FUNCTION_BLOCK fbLightControlV2
		
VAR_INPUT
	bButtonhoofdFunctie				: BOOL;
	bButton2				: BOOL;
	bForceOff			: BOOL;
	bForceOn			: BOOL;

END_VAR
VAR_OUTPUT
	bLight1				: BOOL;
	bLight2				: BOOL;	
	
END_VAR
VAR
	InputTriggerHoofd		: R_trig; 
	InputTrigger2		: R_trig; 
	test:BOOL;
	iCaseVar			:UINT; 
	

	
END_VAR


// This is the first version, ignoring all debounce timers and other issues 
// Base function is a to allow switching a light on and of and having a general reset and general on ( used for construcion)

InputTriggerHoofd(CLK :=  bButtonhoofdFunctie);
InputTrigger2(CLK :=  bButton2);


IF InputTriggerHoofd.Q THEN
	
// ALs alles uit, dan alles aan
	IF (iCaseVar = 0) THEN
		iCaseVar := 1;
	ELSE
		iCaseVar := 0;
	END_IF
END_IF 

IF InputTrigger2.Q THEN
	
	// ALs alles aan, dan de voorste lichten uit
	IF (iCaseVar = 1) THEN
		iCaseVar := 2;
	ELSIF (iCaseVar = 2) THEN
		iCaseVar := 1;
	END_IF
	
END_IF

CASE iCaseVar OF
0:
    bLight1 := FALSE;
	bLight2 := FALSE;
1:
    bLight1 := TRUE;
	bLight2 := TRUE;	
2:
    bLight1 := TRUE;
	bLight2 := FALSE;
3: // eigenlijk niet noodzakelijk
	iCaseVar := 0;
ELSE
	iCaseVar := 0;
END_CASE;




// Deze functie zorgt voor alles aan/Uit Functionaliteit
IF bForceOff THEN
	iCaseVar := 0;
END_IF

IF bForceOn THEN
	iCaseVar := 1;
END_IF

(*function notes: long klick functionality not added, most likley this will be part of another function
This could be a dedicated filter function linked to these functions as needed
*)

END_FUNCTION_BLOCK

(* stored: Version 1.1.0.1, ProductVersion 3.1.4024.11
   POU fbLightControlV2: Id {5790a879-b07f-4e59-b50b-086992a037d0}, SpecialFunc None *)
